(* Schneider Machine Expert - Basic project CutBend, file version 2.6.0.0 *)
(* ProjectInformations: Name=New project *)

HARDWARE
  Cpu 0: TM221CE40R
  EthernetConfiguration: NetworkName=M221, IpAllocationMode=FixedAddress, IpAddress=192.168.0.2, SubnetMask=255.255.255.0
  SerialLineConfiguration: Baud=Baud19200, Parity=ParityEven, DataBits=DataBits8, StopBits=StopBits1, PhysicalMedium=PhysicalMediumRs485, TransmissionMode=TransmissionModeModbusRtu, SlaveId=1, Addressing=SlaveAddressing
  MastTask: UsePeriodScanMode=false, PeriodScan=100
  FastTask: Period=255
  CpuBehavior: StartingMode=StartAsPreviousState, AutoSaveRamOnEeprom=true, WatchdogPeriod=250

SYMBOLS  (address, symbol, comment, settings)
  %M0         "Left Cut Bend"
  %M1         "Manuall"
  %M2         "Rotate"
  %M3         "Rotate Grip"
  %M4         "Component Grip"
  %M5         "Component TF"
  %M6         "Manuall"
  %M7         "System Start"
  %M8         "Polarity Result"
  %M9         "Cut Active"
  %M10        "Cutter Release"
  %M11        "Rotate Active"
  %M12        "Reverse"
  %M13        "Rotate Gripp Release"
  %M20        "M_EMG"
  %M202       "REVERSE"
  %I0.0       "EMG"
  %I0.1       "START"
  %I0.2       "Left Cut FWD"
  %I0.3       "Left Cut BWD"
  %I0.4       "Right Cut FWD"
  %I0.5       "RightCut BWD"
  %I0.6       "Rotate 0"
  %I0.7       "Rotate 1"
  %I0.8       "Rotate Grip Open"
  %I0.9       "Rotate Grip Close"
  %I0.10      "Gripper Comp Open"
  %I0.11      "Gripped Comp Close"
  %I0.12      "Comp TF FWD"
  %I0.13      "Comp TF BWD"
  %I0.14      "BOWL Sensor"
  %I0.15      "Polarity Sensor"
  %I0.18      "Rotate Gripper Open"
  %Q0.0       "Left Cut"
  %Q0.1       "Right Cut"
  %Q0.2       "Rotate"
  %Q0.3       "Rotate Gripper"
  %Q0.4       "TF Comp Grip"
  %Q0.5       "Comp TF"
  %Q0.6       "BOWL FEEDER"

POU New POU
  (* SectionNumber=1 *)

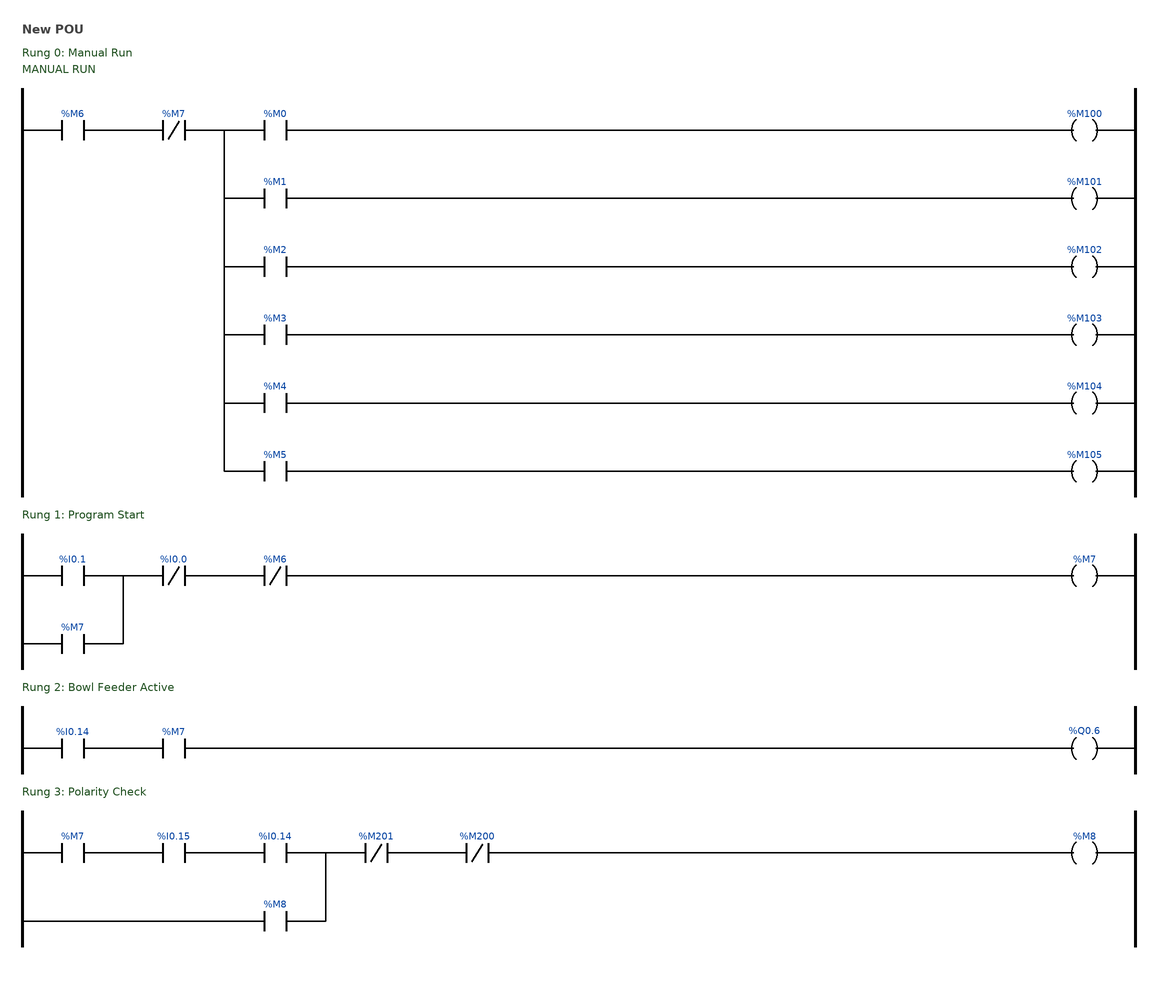

// Rung 0: Manual Run
// MANUAL RUN
  LD %M6
  ANDN %M7
  MPS
  AND %M0
  ST %M100
  MRD
  AND %M1
  ST %M101
  MRD
  AND %M2
  ST %M102
  MRD
  AND %M3
  ST %M103
  MRD
  AND %M4
  ST %M104
  MPP
  AND %M5
  ST %M105
  // as ST:
  //   %M100 := %M6 AND NOT %M7 AND %M0;
  //   %M101 := %M6 AND NOT %M7 AND %M1;
  //   %M102 := %M6 AND NOT %M7 AND %M2;
  //   %M103 := %M6 AND NOT %M7 AND %M3;
  //   %M104 := %M6 AND NOT %M7 AND %M4;
  //   %M105 := %M6 AND NOT %M7 AND %M5;

// Rung 1: Program Start
  LD %I0.1
  OR %M7
  ANDN %I0.0
  ANDN %M6
  ST %M7
  // as ST:
  //   %M7 := (%I0.1 OR %M7) AND NOT %I0.0 AND NOT %M6;

// Rung 2: Bowl Feeder Active
  LD %I0.14
  AND %M7
  ST %Q0.6
  // as ST:
  //   %Q0.6 := %I0.14 AND %M7;

// Rung 3: Polarity Check
  LD %M7
  AND %I0.15
  AND %I0.14
  OR %M8
  ANDN %M201
  ANDN %M200
  ST %M8
  // as ST:
  //   %M8 := (%M7 AND %I0.15 AND %I0.14 OR %M8) AND NOT %M201 AND NOT %M200;

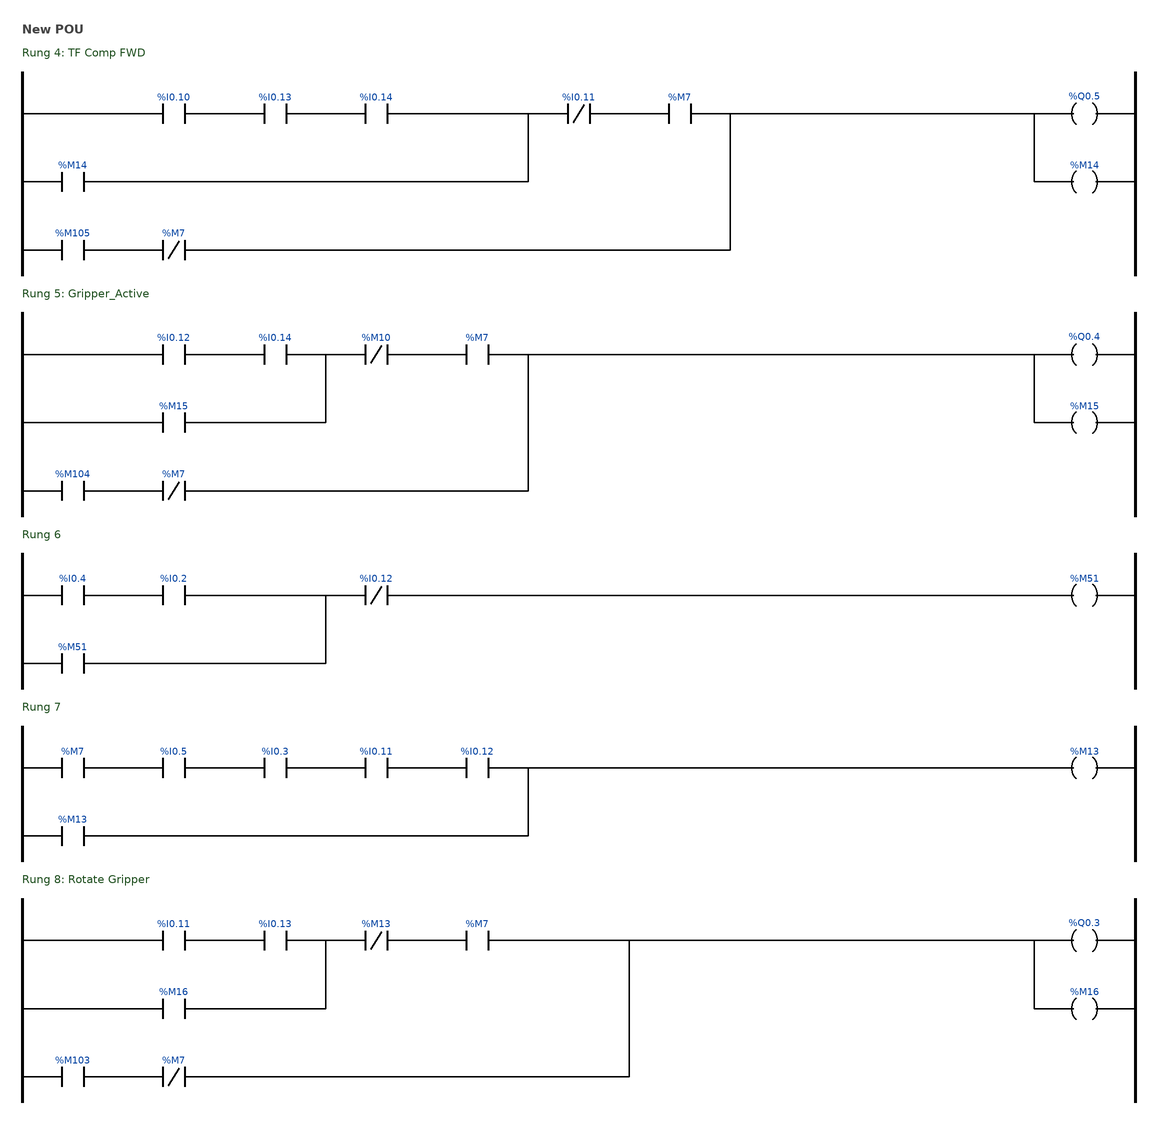

// Rung 4: TF Comp FWD
  LD %I0.10
  AND %I0.13
  AND %I0.14
  OR %M14
  ANDN %I0.11
  AND %M7
  OR( %M105
  ANDN %M7
  )
  ST %Q0.5
  ST %M14
  // as ST:
  //   %Q0.5 := (%I0.10 AND %I0.13 AND %I0.14 OR %M14) AND NOT %I0.11 AND %M7 OR %M105 AND NOT %M7;
  //   %M14 := (%I0.10 AND %I0.13 AND %I0.14 OR %M14) AND NOT %I0.11 AND %M7 OR %M105 AND NOT %M7;

// Rung 5: Gripper_Active
  LD %I0.12
  AND %I0.14
  OR %M15
  ANDN %M10
  AND %M7
  OR( %M104
  ANDN %M7
  )
  ST %Q0.4
  ST %M15
  // as ST:
  //   %Q0.4 := (%I0.12 AND %I0.14 OR %M15) AND NOT %M10 AND %M7 OR %M104 AND NOT %M7;
  //   %M15 := (%I0.12 AND %I0.14 OR %M15) AND NOT %M10 AND %M7 OR %M104 AND NOT %M7;

// Rung 6
  LD %I0.4
  AND %I0.2
  OR %M51
  ANDN %I0.12
  ST %M51
  // as ST:
  //   %M51 := (%I0.4 AND %I0.2 OR %M51) AND NOT %I0.12;

// Rung 7
  LD %M7
  AND %I0.5
  AND %I0.3
  AND %I0.11
  AND %I0.12
  OR %M13
  ST %M13
  // as ST:
  //   %M13 := %M7 AND %I0.5 AND %I0.3 AND %I0.11 AND %I0.12 OR %M13;

// Rung 8: Rotate Gripper
  LD %I0.11
  AND %I0.13
  OR %M16
  ANDN %M13
  AND %M7
  OR( %M103
  ANDN %M7
  )
  ST %Q0.3
  ST %M16
  // as ST:
  //   %Q0.3 := (%I0.11 AND %I0.13 OR %M16) AND NOT %M13 AND %M7 OR %M103 AND NOT %M7;
  //   %M16 := (%I0.11 AND %I0.13 OR %M16) AND NOT %M13 AND %M7 OR %M103 AND NOT %M7;

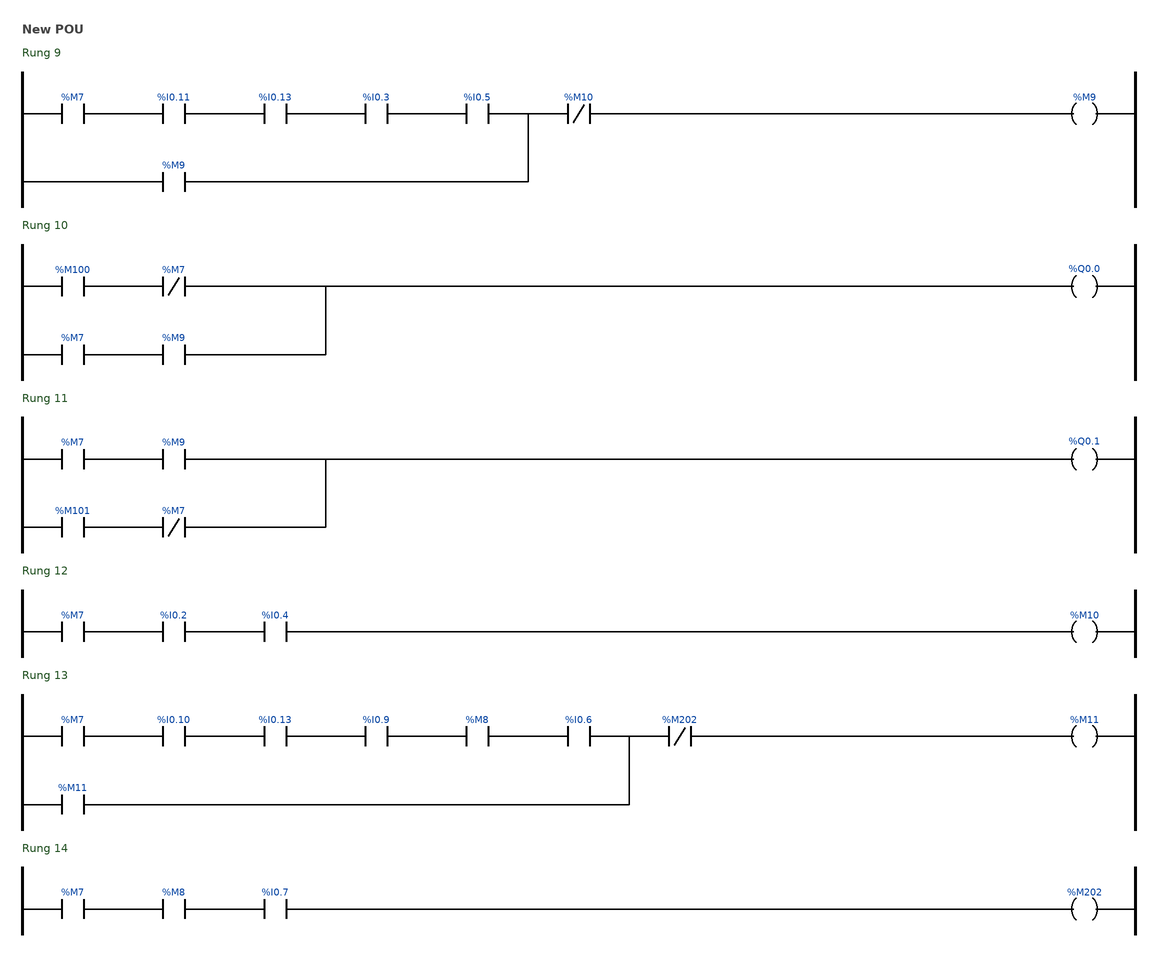

// Rung 9
  LD %M7
  AND %I0.11
  AND %I0.13
  AND %I0.3
  AND %I0.5
  OR %M9
  ANDN %M10
  ST %M9
  // as ST:
  //   %M9 := (%M7 AND %I0.11 AND %I0.13 AND %I0.3 AND %I0.5 OR %M9) AND NOT %M10;

// Rung 10
  LD %M100
  ANDN %M7
  OR( %M7
  AND %M9
  )
  ST %Q0.0
  // as ST:
  //   %Q0.0 := %M100 AND NOT %M7 OR %M7 AND %M9;

// Rung 11
  LD %M7
  AND %M9
  OR( %M101
  ANDN %M7
  )
  ST %Q0.1
  // as ST:
  //   %Q0.1 := %M7 AND %M9 OR %M101 AND NOT %M7;

// Rung 12
  LD %M7
  AND %I0.2
  AND %I0.4
  ST %M10
  // as ST:
  //   %M10 := %M7 AND %I0.2 AND %I0.4;

// Rung 13
  LD %M7
  AND %I0.10
  AND %I0.13
  AND %I0.9
  AND %M8
  AND %I0.6
  OR %M11
  ANDN %M202
  ST %M11
  // as ST:
  //   %M11 := (%M7 AND %I0.10 AND %I0.13 AND %I0.9 AND %M8 AND %I0.6 OR %M11) AND NOT %M202;

// Rung 14
  LD %M7
  AND %M8
  AND %I0.7
  ST %M202
  // as ST:
  //   %M202 := %M7 AND %M8 AND %I0.7;

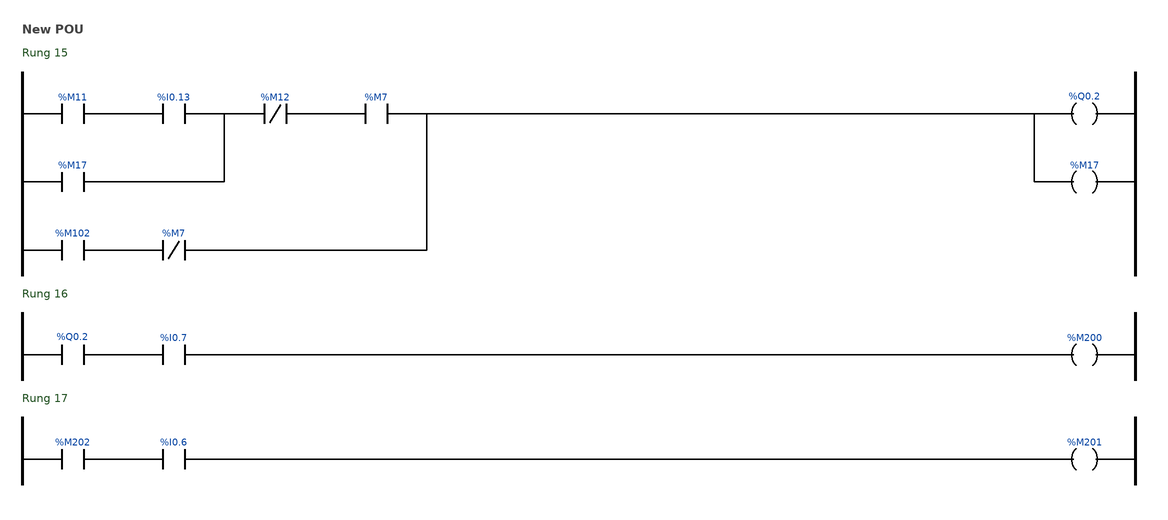

// Rung 15
  LD %M11
  AND %I0.13
  OR %M17
  ANDN %M12
  AND %M7
  OR( %M102
  ANDN %M7
  )
  ST %Q0.2
  ST %M17
  // as ST:
  //   %Q0.2 := (%M11 AND %I0.13 OR %M17) AND NOT %M12 AND %M7 OR %M102 AND NOT %M7;
  //   %M17 := (%M11 AND %I0.13 OR %M17) AND NOT %M12 AND %M7 OR %M102 AND NOT %M7;

// Rung 16
  LD %Q0.2
  AND %I0.7
  ST %M200
  // as ST:
  //   %M200 := %Q0.2 AND %I0.7;

// Rung 17
  LD %M202
  AND %I0.6
  ST %M201
  // as ST:
  //   %M201 := %M202 AND %I0.6;

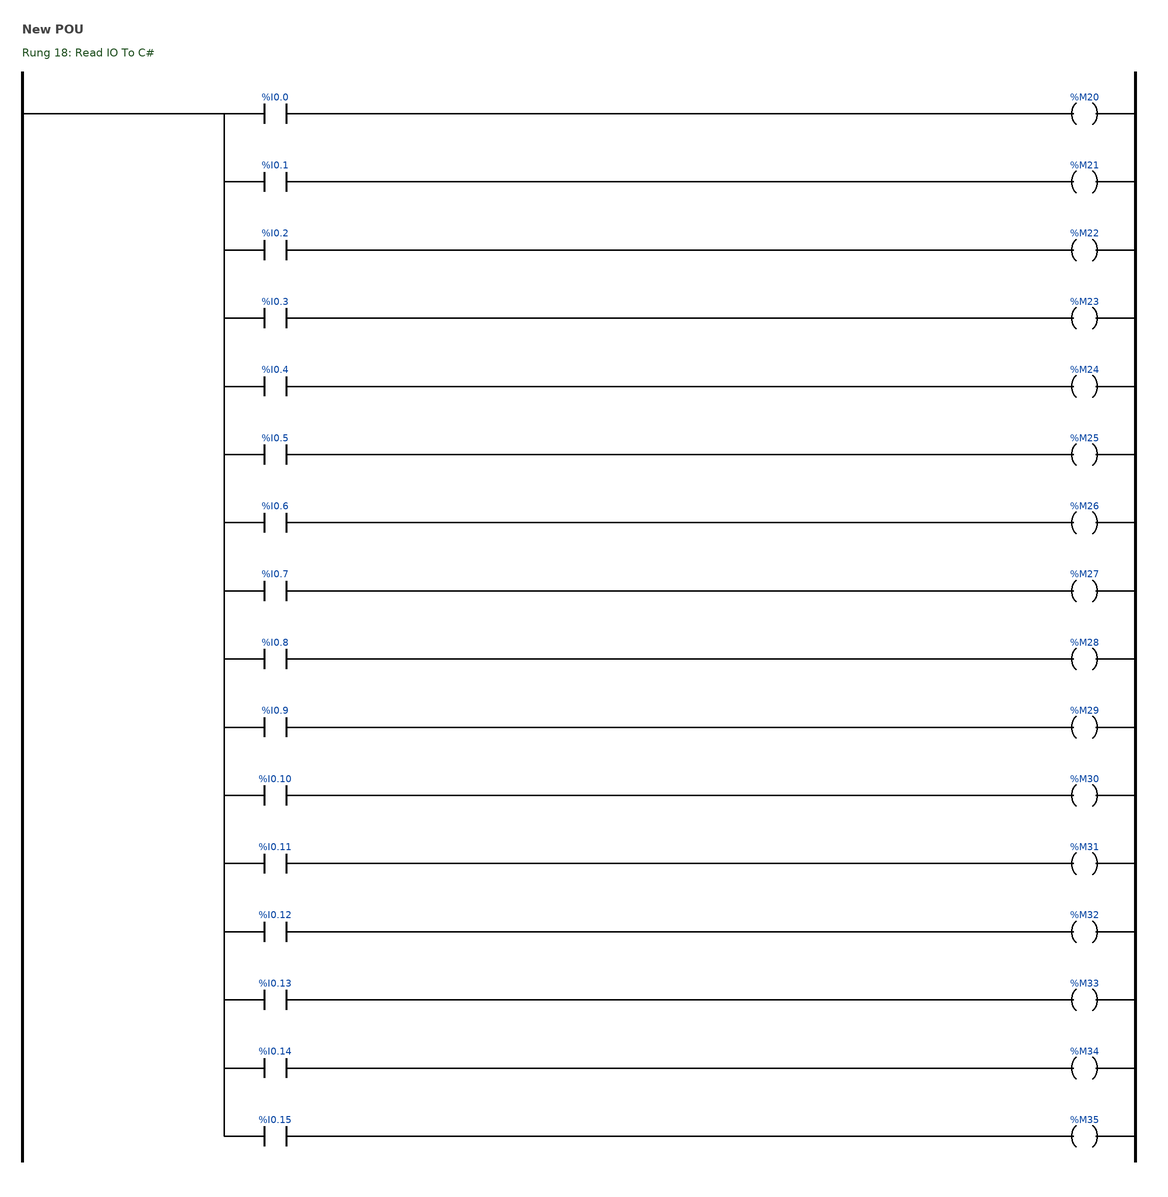

// Rung 18: Read IO To C#
  LD 1
  MPS
  AND %I0.0
  ST %M20
  MRD
  AND %I0.1
  ST %M21
  MRD
  AND %I0.2
  ST %M22
  MRD
  AND %I0.3
  ST %M23
  MRD
  AND %I0.4
  ST %M24
  MRD
  AND %I0.5
  ST %M25
  MRD
  AND %I0.6
  ST %M26
  MRD
  AND %I0.7
  ST %M27
  MRD
  AND %I0.8
  ST %M28
  MRD
  AND %I0.9
  ST %M29
  MRD
  AND %I0.10
  ST %M30
  MRD
  AND %I0.11
  ST %M31
  MRD
  AND %I0.12
  ST %M32
  MRD
  AND %I0.13
  ST %M33
  MRD
  AND %I0.14
  ST %M34
  MPP
  AND %I0.15
  ST %M35
  // as ST:
  //   %M20 := %I0.0;
  //   %M21 := %I0.1;
  //   %M22 := %I0.2;
  //   %M23 := %I0.3;
  //   %M24 := %I0.4;
  //   %M25 := %I0.5;
  //   %M26 := %I0.6;
  //   %M27 := %I0.7;
  //   %M28 := %I0.8;
  //   %M29 := %I0.9;
  //   %M30 := %I0.10;
  //   %M31 := %I0.11;
  //   %M32 := %I0.12;
  //   %M33 := %I0.13;
  //   %M34 := %I0.14;
  //   %M35 := %I0.15;
